INTERFACE ITcoEcatComponent

PROPERTY EcatState : REFERENCE TO TcoEcatSlaveState
GET
END_GET
END_PROPERTY

END_INTERFACE

(* stored: Version 1.1.0.1, ProductVersion 3.1.4024.11
   Itf ITcoEcatComponent: Id {9fd5bf42-1e19-0f6a-2401-12a52f6ad02a}
   Property EcatState: Id {c6113f61-98ce-0c56-30b9-90eddbc9077e}
   Get Get: Id {b587e070-6c6d-0df9-320e-78ebeef1b5e3} *)
